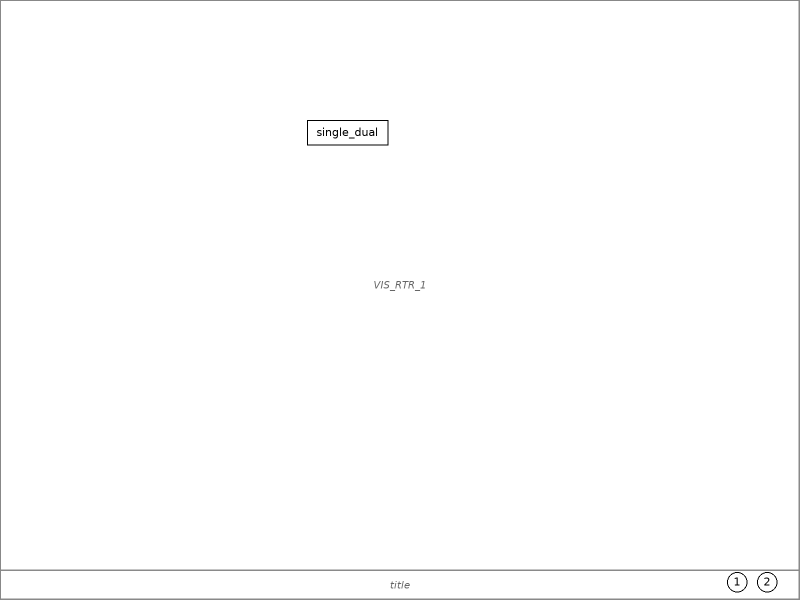
VISUALIZATION F7_RTR  // 800x600
    TabControl (0,0 800x570)
        shows VIS_RTR_1()
        shows VIS_RTR_2()
    RoundedRectangle (307,120 81x25), "single_dual", colour toggle: P_RollToRoll.single_double
    Ellipse (727,572 20x20), "1", colour toggle: stInput.biDualSensor[1]
        toggle stInput.biDualSensor[1]
    Ellipse (757,572 20x20), "2", colour toggle: stInput.biDualSensor[2]
        toggle stInput.biDualSensor[2]
    Frame (0,570 800x30)
        shows title()
END_VISUALIZATION

(* stored: Version 1.1.0.1, ProductVersion 3.1.4024.11
   Visu F7_RTR: Id {0e180b0c-9ffe-4656-9e45-cb51897e2688} *)
